VAR_GLOBAL
	{attribute 'pytmc' := 'pv: AT1L0:GAS:VAC:OVRDON'}
	xSystemOverrideMode	:	BOOL; (* Global system override for the GATT*)
END_VAR

(* stored: Version 1.1.0.1, ProductVersion 3.1.4022.16
   GVL GVL_Variables: Id {13f9e340-d8d3-4a4f-88ba-c53c2f17fe03} *)
